Staubli VAL3: ROBERT_TP6_APPL.pjx

Parameters version=s7.9 stackSize=5000 millimeterUnit=true
Program file=dataAcquisition.pgx
Program file=goToPoint.pgx
Program file=start.pgx
Program file=stop.pgx
Data file=ROBERT_TP6_APPL.dtx
